FUNCTION_BLOCK L2_GEN_Machine (* Composite Function Block Type *)
  (* Standard: 61499-2 *)
  (* Version 0.0, 2015-03-17, EQUEROL, UJI *)
  (* Version 1.0, 2016-01-19, EQUEROL, UJI *)
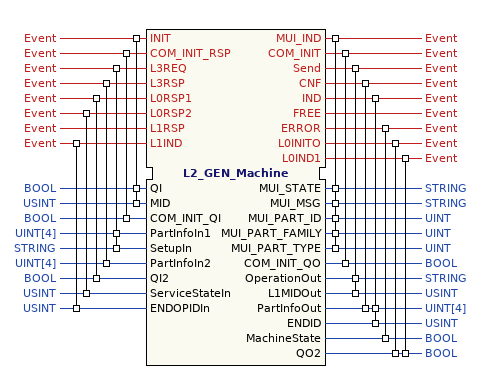
  EVENT_INPUT
    INIT WITH QI, MID; (* Initialization Request *)
    COM_INIT_RSP WITH COM_INIT_QI; (* Communications initialization response *)
    L3REQ WITH PartInfoIn1, SetupIn; (* Setup execution request from layer 3 *)
    L3RSP WITH PartInfoIn2; (* Response from layer 3 *)
    L0RSP1 WITH QI2; (* Layer 0 service response to initialization *)
    L0RSP2 WITH ServiceStateIn; (* Layer 0 service state request response *)
    L1RSP; (* Operation reception confirmation *)
    L1IND WITH ENDOPIDIn; (* Completed OP indication *)
  END_EVENT
  EVENT_OUTPUT
    MUI_IND WITH MUI_STATE, MUI_MSG, MUI_PART_ID, MUI_PART_FAMILY, MUI_PART_TYPE; (* Machine user interface notification *)
    COM_INIT WITH COM_INIT_QO; (* Comunication initialization request *)
    Send WITH OperationOut, L1MIDOut; (* Send operation to Layer 1 *)
    CNF WITH PartInfoOut; (* Assignement reception confirmation *)
    IND WITH PartInfoOut, ENDID; (* completed setup indication *)
    FREE; (* Indicate that the machine is free *)
    ERROR WITH MachineState; (* Indicate a change in the machine state *)
    L0INITO WITH QO2; (* Indicate Service to change state *)
    L0IND1 WITH QO2; (* Request machine service state *)
  END_EVENT
  VAR_INPUT
    QI : BOOL; (* Input event qualifier *)
    MID : USINT; (* Machine identifier *)
    COM_INIT_QI : BOOL; (* Communication initialization qualifier *)
    PartInfoIn1 : ARRAY [0..3] OF UINT; (* Part ID, family, type, MID *)
    SetupIn : STRING; (* Subphase to execute *)
    PartInfoIn2 : ARRAY [0..3] OF UINT; (* ID, Family, Type, MID *)
    QI2 : BOOL; (* Input event qualifier *)
    ServiceStateIn : USINT; (* Machine service state *)
    ENDOPIDIn : USINT; (* Operation end code *)
  END_VAR
  VAR_OUTPUT
    MUI_STATE : STRING; (* String containing the machine's state *)
    MUI_MSG : STRING; (* String containing a message for the MUI *)
    MUI_PART_ID : UINT; (* Current part's ID *)
    MUI_PART_FAMILY : UINT; (* Current part's family *)
    MUI_PART_TYPE : UINT; (* Current part's type *)
    COM_INIT_QO : BOOL; (* Communication initialization qualifier *)
    OperationOut : STRING; (* String containing the serialized operation *)
    L1MIDOut : USINT; (* Layer 1 multicast ID *)
    PartInfoOut : ARRAY [0..3] OF UINT; (* Part identifier, family, type and MID *)
    ENDID : USINT; (* Setup termination code *)
    MachineState : BOOL; (* MachineState *)
    QO2 : BOOL; (* Output event qualifier *)
  END_VAR
  FBS
    L2_ASetupRSPHDLR_1 : L2_ASetupRSPHDLR;
    L2_ExecutionManager_0 : L2_ExecutionManager;
    L2_MachineCore_0 : L2_MachineCore;
    E_DELAY_1 : E_DELAY;
    L2_L1Comm_1 : L2_L1Comm;
    E_DELAY_3 : E_DELAY;
    L2_ASetupREQHDLR_1 : L2_ASetupREQHDLR;
    E_DELAY_2 : E_DELAY;
    L2_StateTracker : L2_StateTracker;
    L2_MachineINIT : L2_MachineINIT;
    E_DELAY : E_DELAY;
    L2_MachineState : L2_MachineState;
  END_FBS
  EVENT_CONNECTIONS
    L2_L1Comm_1.Start TO E_DELAY_1.START;
    L2_ASetupREQHDLR_1.CNF TO L2_MachineCore_0.REQ;
    L2_ASetupREQHDLR_1.INITO TO L2_ASetupRSPHDLR_1.INIT;
    L2_MachineCore_0.stop TO E_DELAY_2.STOP;
    L2_L1Comm_1.Stop TO E_DELAY_1.STOP;
    L2_MachineCore_0.RENEW TO L2_ExecutionManager_0.RENEW;
    L2_ExecutionManager_0.Completed TO L2_MachineCore_0.CompletedSetup;
    E_DELAY_1.EO TO L2_L1Comm_1.Timeout;
    L2_MachineCore_0.start TO E_DELAY_2.START;
    L2_MachineCore_0.NEXT TO L2_ExecutionManager_0.NEXT;
    E_DELAY_2.EO TO L2_MachineCore_0.timeout;
    L2_L1Comm_1.CompletedOP TO L2_MachineCore_0.CompletedOP;
    L2_ASetupRSPHDLR_1.CNF TO L2_MachineCore_0.RSP;
    L2_ExecutionManager_0.ExecuteOP TO L2_L1Comm_1.REQ;
    L2_L1Comm_1.Send TO Send;
    L2_MachineCore_0.CNF TO CNF;
    L2_MachineCore_0.IND TO IND;
    L3REQ TO L2_ASetupREQHDLR_1.REQ;
    L3RSP TO L2_ASetupRSPHDLR_1.RSP;
    L1RSP TO L2_L1Comm_1.RSP;
    L1IND TO L2_L1Comm_1.IND;
    L2_StateTracker.Start TO E_DELAY_3.START;
    L2_StateTracker.Stop TO E_DELAY_3.STOP;
    E_DELAY_3.EO TO L2_StateTracker.Timeout;
    L2_StateTracker.UPDT TO L2_MachineCore_0.UPDT;
    L2_StateTracker.IND TO L0IND1;
    L0RSP2 TO L2_StateTracker.RSP;
    L2_MachineINIT.Start TO E_DELAY.START;
    L2_MachineINIT.Stop TO E_DELAY.STOP;
    E_DELAY.EO TO L2_MachineINIT.TimeOut;
    L2_MachineINIT.L0_INIT TO L0INITO;
    L2_MachineINIT.L2_INIT TO L2_ASetupREQHDLR_1.INIT;
    L2_ASetupRSPHDLR_1.INITO TO L2_ExecutionManager_0.INIT;
    L2_ExecutionManager_0.INITO TO L2_StateTracker.INIT;
    L2_StateTracker.INITO TO L2_MachineINIT.L2_INIT_RSP;
    L0RSP1 TO L2_MachineINIT.L0_INIT_RSP;
    COM_INIT_RSP TO L2_MachineINIT.COM_INIT_RSP;
    L2_MachineINIT.COM_INIT TO COM_INIT;
    INIT TO L2_MachineState.EXT_INIT;
    L2_MachineINIT.IND TO L2_MachineState.M_INIT_RSP;
    L2_MachineCore_0.RENEW TO L2_MachineState.M_BUSY;
    L2_MachineCore_0.FREE TO L2_MachineState.M_FREE;
    L2_MachineCore_0.ERROR TO L2_MachineState.M_ERROR;
    L2_MachineState.M_INIT TO L2_MachineINIT.INIT;
    L2_MachineState.MUI_IND TO MUI_IND;
    L2_MachineState.FREE TO FREE;
    L2_MachineState.ERROR TO ERROR;
  END_CONNECTIONS
  DATA_CONNECTIONS
    L2_ASetupREQHDLR_1.MIDOut TO L2_ASetupRSPHDLR_1.MID;
    L2_L1Comm_1.ENDOPIDOut TO L2_MachineCore_0.ENDOPID;
    L2_ExecutionManager_0.L1MID TO L2_L1Comm_1.L1MIDIn;
    L2_ASetupREQHDLR_1.PartInfoOut TO L2_MachineCore_0.PartInfoIn;
    L2_ExecutionManager_0.ENDSetupID TO L2_MachineCore_0.ENDSetupID;
    L2_ASetupREQHDLR_1.QO TO L2_ASetupRSPHDLR_1.QI;
    L2_ExecutionManager_0.Operation TO L2_L1Comm_1.OperationIn;
    L2_L1Comm_1.Delay TO E_DELAY_1.DT;
    L2_ASetupREQHDLR_1.SetupOut TO L2_ExecutionManager_0.Setup;
    L2_MachineCore_0.NextCode TO L2_ExecutionManager_0.NextCode;
    L2_MachineCore_0.Delay TO E_DELAY_2.DT;
    L2_L1Comm_1.OperationOut TO OperationOut;
    L2_L1Comm_1.L1MIDOut TO L1MIDOut;
    L2_MachineCore_0.PartInfoOut TO PartInfoOut;
    L2_MachineCore_0.ENDID TO ENDID;
    MID TO L2_ASetupREQHDLR_1.MID;
    PartInfoIn1 TO L2_ASetupREQHDLR_1.PartInfoIn;
    SetupIn TO L2_ASetupREQHDLR_1.SetupIn;
    PartInfoIn2 TO L2_ASetupRSPHDLR_1.PartInfo;
    ENDOPIDIn TO L2_L1Comm_1.ENDOPIDIn;
    L2_StateTracker.Delay TO E_DELAY_3.DT;
    L2_StateTracker.ServiceStateOut TO L2_MachineCore_0.ServiceState;
    ServiceStateIn TO L2_StateTracker.ServiceStateIn;
    L2_MachineINIT.TODelay TO E_DELAY.DT;
    L2_MachineINIT.L0_INIT_QO TO QO2;
    L2_MachineINIT.L2_INIT_QO TO L2_ASetupREQHDLR_1.QI;
    L2_ASetupRSPHDLR_1.QO TO L2_ExecutionManager_0.QI;
    L2_ExecutionManager_0.QO TO L2_StateTracker.QI;
    L2_StateTracker.QO TO L2_MachineINIT.L2_INIT_QI;
    QI2 TO L2_MachineINIT.L0_INIT_QI;
    COM_INIT_QI TO L2_MachineINIT.COM_INIT_QI;
    L2_MachineINIT.COM_INIT_QO TO COM_INIT_QO;
    QI TO L2_MachineState.EXT_INIT_QI;
    L2_MachineINIT.INIT_QO TO L2_MachineState.M_INIT_QI;
    L2_MachineINIT.INIT_STATE TO L2_MachineState.M_INIT_STATE;
    L2_MachineCore_0.PartInfoOut TO L2_MachineState.CURRENT_PARTINFO;
    L2_MachineCore_0.MachineState TO L2_MachineState.M_ERROR_STATE;
    L2_MachineState.M_INIT_QO TO L2_MachineINIT.INIT_QI;
    L2_MachineState.MUI_STATE TO MUI_STATE;
    L2_MachineState.MUI_MSG TO MUI_MSG;
    L2_MachineState.MUI_PART_ID TO MUI_PART_ID;
    L2_MachineState.MUI_PART_FAMILY TO MUI_PART_FAMILY;
    L2_MachineState.MUI_PART_TYPE TO MUI_PART_TYPE;
    L2_MachineState.ERROR_STATE TO MachineState;
  END_CONNECTIONS
END_FUNCTION_BLOCK
